// TIA Portal V19 export
VAR_GLOBAL   // PLC tag table "Mixer_Tags"
   Mixer_Start_PB AT %M4.5 : Bool;   // Starts Mixer
   Mixer_Stop_PB AT %M4.6 : Bool;   // Stops Mixer
   Mixer_Hold AT %M4.7 : Bool;   // Mixer held In Running
   Mixer AT %M5.0 : Bool;   // Mixer Status
   "2Hz_Mixer" AT %M4.4 : Bool;   // 2HZ Signal
END_VAR
